PROGRAM Permissives
VAR
	AllChargeRelayClosed 	: BOOL := 0;
	AllDumpRelayOpen		: BOOL := 0;
	ReadyToCharge			: BOOL := 0;
	AllChargerEOC			: BOOL := 0;
	
	//AllCapsDischarged		: BOOL := 0;
	SystemIsSafe			: BOOL := 0;
	
END_VAR

IF LCP1_IO.Segment[1].Module[1].ChargeRly_close = TRUE(*AND all the other modules *) OR HMI_DB.AllChargeRelayCloseBP = TRUE
	THEN
		AllChargeRelayClosed := TRUE;
	ELSE
		AllChargeRelayClosed := FALSE;
END_IF;

IF LCP1_IO.Segment[1].Module[1].DumpRly_open = TRUE(*AND all the other modules *) OR HMI_DB.AllDumpRelaysOpenBP = TRUE
	THEN
		AllDumpRelayOpen := TRUE;
	ELSE
		AllDumpRelayOpen := FALSE;
END_IF;

IF AllChargeRelayClosed = TRUE AND AllDumpRelayOpen = TRUE THEN
	ReadyToCharge := TRUE;
	ELSE 
		ReadyToCharge := FALSE;
END_IF

IF MCP_IO.Charger[1].voltageFeedback <= 10 AND 
	MCP_IO.Charger[1].HV_isON = FALSE AND 
	MCP_IO.Charger[1].inhibited = TRUE AND 
	LCP1_IO.Segment[1].Module[1].DumpRly_open = FALSE
THEN
	(*MCP_IO.Charger[2].voltageFeedback <= 10 AND *)
	SystemIsSafe := TRUE;
	ELSE
		SystemIsSafe := FALSE;
END_IF

IF MCP_IO.Charger[1].EndOfCharge = TRUE AND
	MCP_IO.Charger[2].EndOfCharge = TRUE AND
	MCP_IO.Charger[3].EndOfCharge = TRUE AND
	MCP_IO.Charger[4].EndOfCharge = TRUE AND
	MCP_IO.Charger[5].EndOfCharge = TRUE AND
	MCP_IO.Charger[6].EndOfCharge = TRUE 
THEN
	Permissives_DB.AllChargerEOC := TRUE;
	ELSE
		Permissives_DB.AllChargerEOC := FALSE;

END_IF;

END_PROGRAM

(* stored: Version 1.1.0.1, ProductVersion 3.1.4024.11
   POU Permissives: Id {639d0291-603e-4994-93d7-3ec14345fa0c}, SpecialFunc None *)
